# B&R Automation Studio project project
Automation Studio 4.12.11.2 SP

## Configuration Config2

CPU X20CP3685, AutomationRuntime J4.93, Build 6.3.0, Vc V4.73.5

### Task classes (Cpu.sw)
```
Cyclic#1:
  readcfg <- readcfg.prg
Libraries: operator, runtime, astime, AsIecCon, ArEventLog, FileIO, MyReadCfg, AsBrStr, sys_lib, standard, brsystem
```

### Hardware
```
X20CP3685 : X20CP3685 v1.9.0.0
  Connector IF2:
    ActivateDevice = 1
  ConfigurationID = test_Config2
  Simulation = 1
  FileDevice1
  FileDeviceName1 = USER
  FileDevicePath1 = USER_PATH
```

## Logical view

Binary libraries used (declarations not repeated): operator, runtime, astime, AsIecCon, ArEventLog, FileIO, MyReadCfg, AsBrStr, sys_lib, standard, brsystem

### Program Logical/readcfg

#### Types.typ
```iecst
TYPE
	MachineConfiguration_typ : 	STRUCT
		app_name : STRING[80];
		database_host : STRING[80];
		log_file_path : STRING[80];
		max_connections : DINT;
		port_number : DINT;
		timeout_seconds : DINT;
		buffer_size : DINT;
		debug_mode : BOOL;
		enable_logging : BOOL;
		ssl_enabled : BOOL;
		direction : BOOL;
		cpu_threshold : LREAL;
		memory_limit_gb : LREAL;
	END_STRUCT;
END_TYPE
```

#### Variables.var
```iecst
VAR
	cfgDevice : STRING[32] := 'USER'; (*FileIO device pointing to the USER partition*)
	gMachineCfg : MachineConfiguration_typ;
	cfgFileName : STRING[80] := 'settings.ini';
	cfgIdent : UDINT;
	content : STRING[4096];
	last_error : DINT;
	key_exist : BOOL;
END_VAR
```

#### Main.st
```iecst
PROGRAM _INIT
	cfgIdent := MRC_Open(ADR(cfgDevice), ADR(cfgFileName));

	(* check if key exist *)
	key_exist := MRC_KeyExists( cfgIdent, ADR('app_name') );

	(* read STRING *)
	MRC_ReadSTRING( cfgIdent, ADR('app_name'), ADR(gMachineCfg.app_name), SIZEOF(gMachineCfg.app_name), ADR('<unknown>') );
	MRC_ReadSTRING( cfgIdent, ADR('database_host'), ADR(gMachineCfg.database_host), SIZEOF(gMachineCfg.database_host), ADR('0.0.0.0') );
	MRC_ReadSTRING( cfgIdent, ADR('log_file_path'), ADR(gMachineCfg.log_file_path), SIZEOF(gMachineCfg.log_file_path), ADR('\') );

	(* read DINT *)
	gMachineCfg.max_connections := MRC_ReadDINT(cfgIdent, ADR('max_connections'), 0);
	gMachineCfg.port_number := MRC_ReadDINT(cfgIdent, ADR('port_number'), 0);
	gMachineCfg.timeout_seconds := MRC_ReadDINT(cfgIdent, ADR('timeout_seconds'), 0);
	gMachineCfg.buffer_size := MRC_ReadDINT(cfgIdent, ADR('buffer_size'), 0);

	(* read BOOL *)
	gMachineCfg.debug_mode := MRC_ReadBOOL(cfgIdent, ADR('debug_mode'), FALSE);
	gMachineCfg.enable_logging := MRC_ReadBOOL(cfgIdent, ADR('enable_logging'), FALSE);
	gMachineCfg.ssl_enabled := MRC_ReadBOOL(cfgIdent, ADR('ssl_enabled'), FALSE);
	gMachineCfg.direction := MRC_ReadBOOL(cfgIdent, ADR('direction'), FALSE);

	(* read LREAL *)
	gMachineCfg.cpu_threshold := MRC_ReadLREAL(cfgIdent, ADR('cpu_threshold'), 0.0);
	gMachineCfg.memory_limit_gb := MRC_ReadLREAL(cfgIdent, ADR('memory_limit_gb'), 0.0);

	(* read complete file content *)
	MRC_ReadContent( cfgIdent, ADR(content), SIZEOF(content) );

	(* read not existing key *)
	gMachineCfg.ssl_enabled := MRC_ReadBOOL(cfgIdent, ADR('not_exist'), FALSE);
	last_error := MRC_GetLastError(cfgIdent); (* returns MRC_ERR_KEY_NOT_FOUND *)

	MRC_Close(cfgIdent);
	cfgIdent := 0;

	ST_tmp_suspend(0);
END_PROGRAM

PROGRAM _CYCLIC

END_PROGRAM

PROGRAM _EXIT
	IF cfgIdent <> 0 THEN
		MRC_Close(cfgIdent);
		cfgIdent := 0;
	END_IF
END_PROGRAM
```
